{attribute wpf [Container(Layout.Tabs)]}
TYPE
    TechnologyComponents EXTENDS TcoCore.TcoStruct :
    STRUCT
      	{attribute wpf [Container(Layout.Stack)]}
        {attribute addProperty Name "<#Presure OK #>"}
        AirPresureOk : TcoElements.TcoDi(THISSTRUCT);  
	
		{attribute wpf [Container(Layout.Stack)]}
        {attribute addProperty Name "<#Emergency Stop  #>"}
        EmergencyStop : TcoEmergencyStop(THISSTRUCT);

		{attribute wpf [Container(Layout.Stack)]}
        {attribute addProperty Name "<#Global control voltage  #>"}
        GlobalControlVoltage : TcoControlVoltage(THISSTRUCT);
		
		{attribute wpf [Container(Layout.Stack)]}
        {attribute addProperty Name "<#Local control voltage  #>"}
        LocalControlVoltage : TcoControlVoltage(THISSTRUCT);
		
		{attribute wpf [Container(Layout.Stack)]}
        {attribute addProperty Name "<#Local door voltage  #>"}
        LocalDoorVoltage : TcoControlVoltage(THISSTRUCT);
		
		
		{attribute wpf [Container(Layout.Stack)]}
        {attribute addProperty Name "<#Control Buttons #>"}
        ControlButtons : TcoControlButtons(THISSTRUCT);
		
        {attribute addProperty Name "<#Mode key #>"}
        ModeKey : TcoKeyMode(THISSTRUCT);
		
		{attribute addProperty Name "<#Normal/Service key #>"}
        NormalServiceKey : TcoKeyNormalService(THISSTRUCT);
		
		
		{attribute addProperty Name "<#Door#>"}
        Door : TcoDoor(THISSTRUCT);

		{attribute addProperty Name "<#Key door#>"}
        DoorKey : TcoKeyDoor(THISSTRUCT);

		
		
		{attribute wpf [Container(Layout.Stack)]}
        {attribute addProperty Name "<#Door circuit #>"}
        DoorCicuit : TcoDoorCircuit(THISSTRUCT);

		
		{attribute wpf [Container(Layout.Stack)]}
        {attribute addProperty Name "<#Zone #>"}
        Zone : TcoControlledZone(THISSTRUCT);



    END_STRUCT
END_TYPE

(* stored: Version 1.1.0.1
   DUT TechnologyComponents: Id {c8b41d55-fe8d-4b4c-a14b-49ecddfbf052} *)
